{attribute 'GeneratedUsingTerminal: EK1100-0000-0018'}
{attribute addProperty BoxType "EK1100-0000-0018"}
{attribute addProperty Id "Beckhoff_ER6xxxEK1122Beckhoff_ER6xxxEK1122_AE47C095446"}
{attribute addProperty CRC "2054056739"}
{attribute addProperty Size "446"}
TYPE Beckhoff_ER6xxx_7A6E6B23 EXTENDS EK1100_AB5A9467 :
STRUCT
	{attribute addProperty Name "Beckhoff_ER6xxxEK1122"}
	{attribute addProperty PreviousPort "Beckhoff ER6xxx : B"}
	Beckhoff_ER6xxxEK1122 : Beckhoff_ER6xxxEK1122_AE47C095;
END_STRUCT
END_TYPE

(* stored: Version 1.2.0.0, ProductVersion 3.1.4024.9
   DUT Beckhoff_ER6xxx_7A6E6B23: Id {b255b415-c35e-4697-9d1f-ba1d1a3d3432} *)
